{region '#Template'}
	{attribute 'Category' := 'AC'}
	{attribute 'Version' := '0.0.1.0'}
	{attribute 'Tags' := 'AC, General'}
	{attribute 'Description' := 'Betriebsart 1 stufig	// Operating mode 1 stufig'}
{endregion}
FUNCTION_BLOCK FB_BA_AC_OpMod1St EXTENDS FB_BA_View
VAR_INPUT
	bSmExttSuA				: BOOL;	// smoke extraction supply air
	bSmExttExhA				: BOOL;	// smoke extraction exhaust air
	bFireDetc				: BOOL;	// fire detection alarm
	bForcVent				: BOOL;	// Forced ventilation
	bEmgOff					: BOOL;	// emergency stop
	bFrst					: BOOL;	// Frost protection is active
	bCentSwiOff				: BOOL;	// Central switch-off	
	bAlmShutOff				: BOOL;	// Shut Off plant collective alarm
	bNgtCol					: BOOL;	// Summer night cooling
	bColDwnPrtc				: BOOL;	// Cooling down protection
	bOvrHtgPrtc				: BOOL;	// Overheating protection
END_VAR
VAR_OUTPUT
	eOpMode					: E_BA_AC_OpMod01;
END_VAR
VAR_INPUT CONSTANT
	OpModMan				: FB_BA_MV_Op;	
	Sched					: FB_BA_SchedM;
	OpModPr					: FB_BA_MV_Op;
END_VAR
VAR
	PrioSwi					: FB_BA_PrioSwi_UDI24;
END_VAR

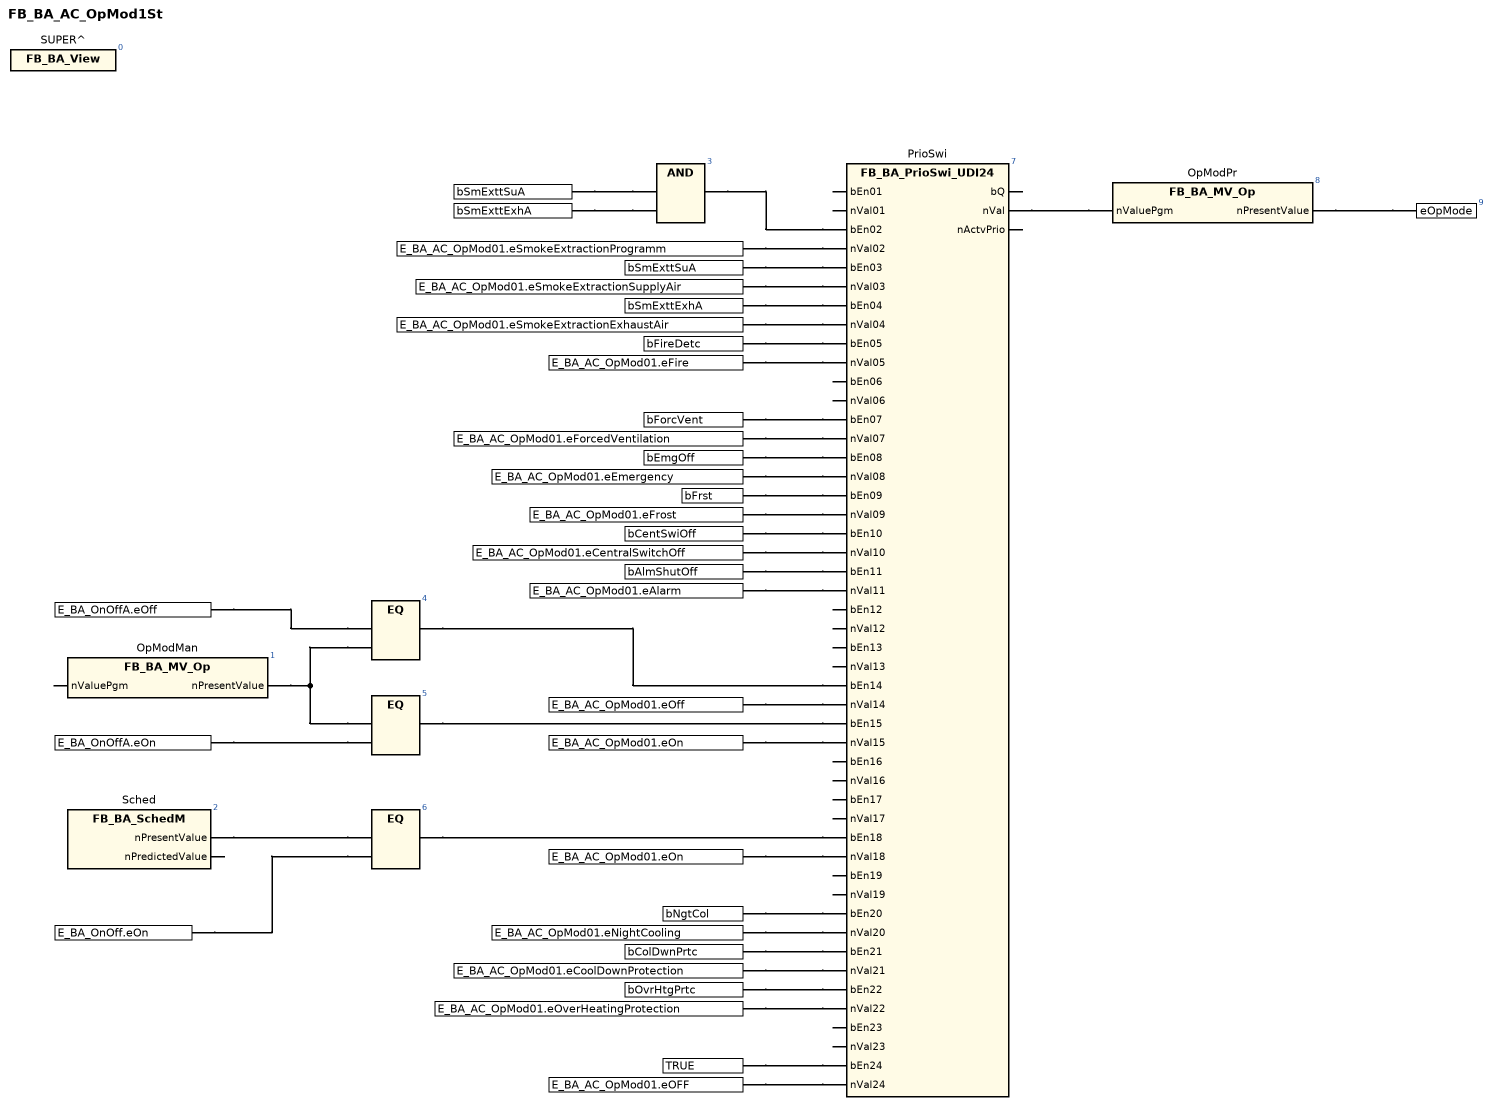
SUPER^(); // FB_BA_View
OpModMan(); // FB_BA_MV_Op
Sched(); // FB_BA_SchedM
PrioSwi(
    bEn02 := bSmExttSuA AND bSmExttExhA,
    nVal02 := E_BA_AC_OpMod01.eSmokeExtractionProgramm,
    bEn03 := bSmExttSuA,
    nVal03 := E_BA_AC_OpMod01.eSmokeExtractionSupplyAir,
    bEn04 := bSmExttExhA,
    nVal04 := E_BA_AC_OpMod01.eSmokeExtractionExhaustAir,
    bEn05 := bFireDetc,
    nVal05 := E_BA_AC_OpMod01.eFire,
    bEn07 := bForcVent,
    nVal07 := E_BA_AC_OpMod01.eForcedVentilation,
    bEn08 := bEmgOff,
    nVal08 := E_BA_AC_OpMod01.eEmergency,
    bEn09 := bFrst,
    nVal09 := E_BA_AC_OpMod01.eFrost,
    bEn10 := bCentSwiOff,
    nVal10 := E_BA_AC_OpMod01.eCentralSwitchOff,
    bEn11 := bAlmShutOff,
    nVal11 := E_BA_AC_OpMod01.eAlarm,
    bEn14 := E_BA_OnOffA.eOff = OpModMan.nPresentValue,
    nVal14 := E_BA_AC_OpMod01.eOff,
    bEn15 := OpModMan.nPresentValue = E_BA_OnOffA.eOn,
    nVal15 := E_BA_AC_OpMod01.eOn,
    bEn18 := Sched.nPresentValue = E_BA_OnOff.eOn,
    nVal18 := E_BA_AC_OpMod01.eOn,
    bEn20 := bNgtCol,
    nVal20 := E_BA_AC_OpMod01.eNightCooling,
    bEn21 := bColDwnPrtc,
    nVal21 := E_BA_AC_OpMod01.eCoolDownProtection,
    bEn22 := bOvrHtgPrtc,
    nVal22 := E_BA_AC_OpMod01.eOverHeatingProtection,
    bEn24 := TRUE,
    nVal24 := E_BA_AC_OpMod01.eOFF); // FB_BA_PrioSwi_UDI24
OpModPr(nValuePgm := PrioSwi.nVal); // FB_BA_MV_Op
eOpMode := OpModPr.nPresentValue;

METHOD EvaluateOpMode
VAR_INPUT
	nOpMode				: UDINT;
	nOffMode			: UDINT;				// Index of operation mode [Off]
END_VAR
VAR_OUTPUT
	bQ					: BOOL;
	ePltOpMode			: E_BA_AC_OpMod01;
END_VAR
VAR_INST
	{attribute 'hide'}
	{attribute 'no_copy'}
	_iStateObj			: I_BA_MultistateObject;
	{attribute 'hide'}
	{attribute 'no_copy'}
	_nOffset			: UDINT;
END_VAR
VAR
	_iObj				: I_BA_Object;
END_VAR
VAR CONSTANT
	OP_MODE_SUBJECT		: T_BA_MedString		:= 'Sched';
END_VAR
// Initialization:
IF (_iStateObj = 0) AND_THEN (State = E_BA_ObjectState.ePostInit) THEN
	// Obtain operation mode objects:
	IF (QueryObjectPrf(OP_MODE_SUBJECT, 0, iResult=>_iObj)) AND_THEN (__QUERYINTERFACE(_iObj, _iStateObj)) THEN
		// Determine plant operation mode corresponding to object's operation mode:
		CASE (_iStateObj.StateCount) OF
			2:		_nOffset := (E_BA_AC_OpMod01.eOn-E_BA_AC_OpMod01.eOn);			// Assuming [Off,On]:
			3,4:	_nOffset := (E_BA_AC_OpMod01.eStep1-E_BA_AC_OpMod01.eOn);		// Assuming [Off,Step1,Step2,Step3]:
		ELSE
			_sTemp := _iStateObj.InstDescription;
			LogMsg.Show1(ADSLOG_MSGTYPE_ERROR, 'EOM24', 'Failed to determine plant operation mode due to unexpected state count of "%d"!', F_STRINGEx(_sTemp), FALSE);
			_iStateObj := 0;
			RETURN;
		END_CASE
	ELSE
		_sTemp := OP_MODE_PROFILE.ProfileName;
		fbLogMsg.Show1(ADSLOG_MSGTYPE_ERROR, 'GPOM04', 'Failed to determine plant operation mode because object with profile "%s" could not be found!', F_STRINGEx(OP_MODE_SUBJECT), FALSE);
	END_IF
END_IF

// Determinate plant operation mode:
IF (_iStateObj = 0) OR_ELSE (_iStateObj.State <> E_BA_ObjectState.eOperation) THEN
	ePltOpMode := E_BA_AC_OpMod01.Invalid;
ELSE
	IF (nOpMode < 1) THEN
		// No operation mode commanded:
		ePltOpMode := E_BA_AC_OpMod01.Invalid;
	ELSIF (nOpMode = 1) THEN
		// Default operation mode commanded (Skip):
		ePltOpMode := E_BA_AC_OpMod01.Invalid;
	ELSE
		ePltOpMode := (E_BA_AC_OpMod01.eOff + _nOffset + (nOpMode-nOffMode));
	END_IF
END_IF

// Validate result:
IF (ePltOpMode = E_BA_AC_OpMod01.Invalid) THEN
	bQ := FALSE;
	ePltOpMode := E_BA_AC_OpMod01.eOff;
ELSE
	bQ := TRUE;
END_IF
END_METHOD

METHOD FB_init : BOOL
VAR_INPUT
	bInitRetains : BOOL; // if TRUE, the retain variables are initialized (warm start / cold start)
	bInCopyCode : BOOL;  // if TRUE, the instance afterwards gets moved into the copy code (online change)
END_VAR
OpModMan.iParent			:= THIS^;
OpModMan.iLabel				:= LblCmpAC.General_OpModMan;							
OpModMan.sObjectName		:= '{Idx=01}';								 	 
OpModMan.aStateText[1]		:= Texts.txtAuto;
OpModMan.aStateText[2]		:= Texts.txtOff;
OpModMan.aStateText[3]		:= Texts.txtOn;
OpModMan.nValueRm			:= E_BA_OnOffA.eAutomatic;

OpModPr.iParent				:= THIS^;
OpModPr.iLabel				:= LblCmpAC.General_OpModPr;							
OpModPr.sObjectName			:= '{Idx=01}';								 	 
OpModPr.aStateText[1]		:= Texts.txtOff;
OpModPr.aStateText[2]		:= Texts.txtOn;
OpModPr.aStateText[3]		:= Texts.txtEmergencyStop;
OpModPr.aStateText[4]		:= Texts.txtFrost;
OpModPr.aStateText[5]		:= Texts.txtSmokeExtraction_P;
OpModPr.aStateText[6]		:= Texts.txtSmokeExtractionSupplyAir;
OpModPr.aStateText[7]		:= Texts.txtSmokeExtractionExtractAir;
OpModPr.aStateText[8]		:= Texts.txtFire;
OpModPr.aStateText[9]		:= Texts.txtNightCooling;
OpModPr.aStateText[10]		:= Texts.txtCoolDownProtection;
OpModPr.aStateText[11]		:= Texts.txtOverHeatingProtection;
OpModPr.aStateText[12]		:= Texts.txtDisturb;
OpModPr.aStateText[13]		:= Texts.txtForcedVentilation;
OpModPr.aStateText[14]		:= Texts.txtCentralSwitchOff; 		

Sched.iParent											:= THIS^;
Sched.iLabel											:= LblCmpAC.General_Sched;							
Sched.sObjectName										:= '{Idx=01}';		
Sched.aStateText[1]										:= Texts.txtOff;
Sched.aStateText[2]										:= Texts.txtOn;
Sched.nPredictTime										:= 0;
Sched.nDefaultValue										:= E_BA_OnOff.eOff;
Sched.bWriteWeekly										:= FALSE;
//	Monday
Sched.aWeek[E_BA_Weekday.eMonday,1].eState				:= E_BA_SchedEntryState.eValue;
Sched.aWeek[E_BA_Weekday.eMonday,1].uValue.udiVal		:= E_BA_OnOff.eOn;
Sched.aWeek[E_BA_Weekday.eMonday,1].stTime.nHour		:= 6;
Sched.aWeek[E_BA_Weekday.eMonday,1].stTime.nMinute		:= 0;
Sched.aWeek[E_BA_Weekday.eMonday,1].stTime.nSecond		:= 0;
Sched.aWeek[E_BA_Weekday.eMonday,2].eState				:= E_BA_SchedEntryState.eValue;
Sched.aWeek[E_BA_Weekday.eMonday,2].uValue.udiVal		:= E_BA_OnOff.eOff;
Sched.aWeek[E_BA_Weekday.eMonday,2].stTime.nHour		:= 20;
Sched.aWeek[E_BA_Weekday.eMonday,2].stTime.nMinute		:= 0;
Sched.aWeek[E_BA_Weekday.eMonday,2].stTime.nSecond		:= 0;
Sched.aWeek[E_BA_Weekday.eMonday,3].eState				:= E_BA_SchedEntryState.eValue;
Sched.aWeek[E_BA_Weekday.eMonday,3].uValue.udiVal		:= E_BA_OnOff.eOff;
Sched.aWeek[E_BA_Weekday.eMonday,3].stTime.nHour		:= 0;
Sched.aWeek[E_BA_Weekday.eMonday,3].stTime.nMinute		:= 0;
Sched.aWeek[E_BA_Weekday.eMonday,3].stTime.nSecond		:= 0;
//	Tuesday
Sched.aWeek[E_BA_Weekday.eTuesday,1].eState				:= E_BA_SchedEntryState.eValue;
Sched.aWeek[E_BA_Weekday.eTuesday,1].uValue.udiVal		:= E_BA_OnOff.eOn;
Sched.aWeek[E_BA_Weekday.eTuesday,1].stTime.nHour		:= 6;
Sched.aWeek[E_BA_Weekday.eTuesday,1].stTime.nMinute		:= 0;
Sched.aWeek[E_BA_Weekday.eTuesday,1].stTime.nSecond		:= 0;
Sched.aWeek[E_BA_Weekday.eTuesday,2].eState				:= E_BA_SchedEntryState.eValue;
Sched.aWeek[E_BA_Weekday.eTuesday,2].uValue.udiVal		:= E_BA_OnOff.eOff;
Sched.aWeek[E_BA_Weekday.eTuesday,2].stTime.nHour		:= 20;
Sched.aWeek[E_BA_Weekday.eTuesday,2].stTime.nMinute		:= 0;
Sched.aWeek[E_BA_Weekday.eTuesday,2].stTime.nSecond		:= 0;
Sched.aWeek[E_BA_Weekday.eTuesday,3].eState				:= E_BA_SchedEntryState.eValue;
Sched.aWeek[E_BA_Weekday.eTuesday,3].uValue.udiVal		:= E_BA_OnOff.eOff;
Sched.aWeek[E_BA_Weekday.eTuesday,3].stTime.nHour		:= 0;
Sched.aWeek[E_BA_Weekday.eTuesday,3].stTime.nMinute		:= 0;
Sched.aWeek[E_BA_Weekday.eTuesday,3].stTime.nSecond		:= 0;
//	Wednesday
Sched.aWeek[E_BA_Weekday.eWednesday,1].eState			:= E_BA_SchedEntryState.eValue;
Sched.aWeek[E_BA_Weekday.eWednesday,1].uValue.udiVal	:= E_BA_OnOff.eOn;
Sched.aWeek[E_BA_Weekday.eWednesday,1].stTime.nHour		:= 6;
Sched.aWeek[E_BA_Weekday.eWednesday,1].stTime.nMinute	:= 0;
Sched.aWeek[E_BA_Weekday.eWednesday,1].stTime.nSecond	:= 0;
Sched.aWeek[E_BA_Weekday.eWednesday,2].eState			:= E_BA_SchedEntryState.eValue;
Sched.aWeek[E_BA_Weekday.eWednesday,2].uValue.udiVal	:= E_BA_OnOff.eOff;
Sched.aWeek[E_BA_Weekday.eWednesday,2].stTime.nHour		:= 20;
Sched.aWeek[E_BA_Weekday.eWednesday,2].stTime.nMinute	:= 0;
Sched.aWeek[E_BA_Weekday.eWednesday,2].stTime.nSecond	:= 0;
Sched.aWeek[E_BA_Weekday.eWednesday,3].eState			:= E_BA_SchedEntryState.eValue;
Sched.aWeek[E_BA_Weekday.eWednesday,3].uValue.udiVal	:= E_BA_OnOff.eOff;
Sched.aWeek[E_BA_Weekday.eWednesday,3].stTime.nHour		:= 0;
Sched.aWeek[E_BA_Weekday.eWednesday,3].stTime.nMinute	:= 0;
Sched.aWeek[E_BA_Weekday.eWednesday,3].stTime.nSecond	:= 0;
//	Thursday
Sched.aWeek[E_BA_Weekday.eThursday,1].eState			:= E_BA_SchedEntryState.eValue;
Sched.aWeek[E_BA_Weekday.eThursday,1].uValue.udiVal		:= E_BA_OnOff.eOn;
Sched.aWeek[E_BA_Weekday.eThursday,1].stTime.nHour		:= 6;
Sched.aWeek[E_BA_Weekday.eThursday,1].stTime.nMinute	:= 0;
Sched.aWeek[E_BA_Weekday.eThursday,1].stTime.nSecond	:= 0;
Sched.aWeek[E_BA_Weekday.eThursday,2].eState			:= E_BA_SchedEntryState.eValue;
Sched.aWeek[E_BA_Weekday.eThursday,2].uValue.udiVal		:= E_BA_OnOff.eOff;
Sched.aWeek[E_BA_Weekday.eThursday,2].stTime.nHour		:= 20;
Sched.aWeek[E_BA_Weekday.eThursday,2].stTime.nMinute	:= 0;
Sched.aWeek[E_BA_Weekday.eThursday,2].stTime.nSecond	:= 0;
Sched.aWeek[E_BA_Weekday.eThursday,3].eState			:= E_BA_SchedEntryState.eValue;
Sched.aWeek[E_BA_Weekday.eThursday,3].uValue.udiVal		:= E_BA_OnOff.eOff;
Sched.aWeek[E_BA_Weekday.eThursday,3].stTime.nHour		:= 0;
Sched.aWeek[E_BA_Weekday.eThursday,3].stTime.nMinute	:= 0;
Sched.aWeek[E_BA_Weekday.eThursday,3].stTime.nSecond	:= 0;
//	Friday
Sched.aWeek[E_BA_Weekday.eFriday,1].eState				:= E_BA_SchedEntryState.eValue;
Sched.aWeek[E_BA_Weekday.eFriday,1].uValue.udiVal		:= E_BA_OnOff.eOn;
Sched.aWeek[E_BA_Weekday.eFriday,1].stTime.nHour		:= 6;
Sched.aWeek[E_BA_Weekday.eFriday,1].stTime.nMinute		:= 0;
Sched.aWeek[E_BA_Weekday.eFriday,1].stTime.nSecond		:= 0;
Sched.aWeek[E_BA_Weekday.eFriday,2].eState				:= E_BA_SchedEntryState.eValue;
Sched.aWeek[E_BA_Weekday.eFriday,2].uValue.udiVal		:= E_BA_OnOff.eOff;
Sched.aWeek[E_BA_Weekday.eFriday,2].stTime.nHour		:= 20;
Sched.aWeek[E_BA_Weekday.eFriday,2].stTime.nMinute		:= 0;
Sched.aWeek[E_BA_Weekday.eFriday,2].stTime.nSecond		:= 0;
Sched.aWeek[E_BA_Weekday.eFriday,3].eState				:= E_BA_SchedEntryState.eValue;
Sched.aWeek[E_BA_Weekday.eFriday,3].uValue.udiVal		:= E_BA_OnOff.eOff;
Sched.aWeek[E_BA_Weekday.eFriday,3].stTime.nHour		:= 0;
Sched.aWeek[E_BA_Weekday.eFriday,3].stTime.nMinute		:= 0;
Sched.aWeek[E_BA_Weekday.eFriday,3].stTime.nSecond		:= 0;
Sched.bWriteException									:= FALSE;
END_METHOD

END_FUNCTION_BLOCK

(* stored: Version 1.1.0.1, ProductVersion 3.1.4024.6
   POU FB_BA_AC_OpMod1St: Id {5aa242a4-a3ec-4579-82a3-719c4d0ceafb}, SpecialFunc None
   Folder Management: Id {64ab1b7c-7b06-4624-86f3-e4d66fc3ca92}
   Method EvaluateOpMode: Id {00dbc6a4-a0b3-428f-afe6-31202c4ea923}
   Method FB_init: Id {8ab81cca-7537-4e59-8205-768ab224e1bf} *)
